// TIA Portal V19 export
DATA_BLOCK "MC_MoveAbsolute_DB"   // DB9
// stored: InstanceOfName MC_MoveAbsolute, OfSystemLibElement MC_MoveAbsolute, OfSystemLibVersion 7.0
"MC_MoveAbsolute"
   // VAR_INPUT
   //    Axis : TO_PositioningAxis;
   //    Execute : Bool;
   //    Position : Real;
   //    Velocity : Real;
   //    Direction : Int;
   // END_VAR
   // VAR_OUTPUT
   //    Done : Bool;
   //    Busy : Bool;
   //    CommandAborted : Bool;
   //    Error : Bool;
   //    ErrorID : Word;
   //    ErrorInfo : Word;
   // END_VAR
   // VAR
   //    FB_ID : DInt;
   // END_VAR
BEGIN
END_DATA_BLOCK
